# EPICS substitutions: db/ecmcIPOS4808_AUX.substitutions
file ecmcIPOSXXXX_AUX.template
{
	pattern {CURRESLO}
		{6.105e-4}
}
